(* CoDeSys 2.3.9.47 project: mqtt.pro *)
(* Libraries: C:\Program Files\WAGO Software\CoDeSys V2.3\Targets\WAGO\Libraries\32_Bit\oscat_basic_333.lib 9.2.16 17:15:54, SysLibSockets.lib 22.5.14 15:16:32, WagoLibEthernet_01.lib 11.2.16 17:05:44, Standard.lib 20.5.14 07:13:26, Iecsfc.lib 16.5.13 13:00:50, SYSLIBCALLBACK.LIB 16.5.13 13:00:50 *)

(* PLC configuration (modules and I/O channels)
K-Bus [K_Bus] node 0, in %IB0 out %QB0 {KbusBusMode = 1; KbusCycleTime = 10000; KbusThreadPriority = 0; KbusSetOutputsToZeroOnApplicationStop = 1}
Modbus variables [PFC200MODBUS] node 1, in %IB0 out %QB0 {PlcStopBehaviour = 1; FiledbusErrorBehaviour = 1; TcpOperation = 1; TcpPort = 502; TcpTimeout = 600; UdpOperation = 1; UdpPort = 502; RtuOperation = 0; NodeId = 1; ResponseTimeout = 5000; Interface = 0; Baud = 115200; StopBits = 1; Parity = 1; FlowCtrl = 0; PhysInterface = 0}
unused [PFC200CANOPEN_UNUSED] node 2, in %IB6000 out %QB6000
Modbus-Master [MB_MASTER] node 3, in %IB0 out %QB0
*)

(* Task configuration *)
TASK Schedule (PRIORITY := 31, INTERVAL := T#100ms);
	PLC_PRG();
END_TASK

(* Global variable list: Globale_Variablen *)
VAR_GLOBAL
	xxSubscribe: BOOL := TRUE;
	xxPublish : BOOL     := TRUE;
	SubPubState : INT;
END_VAR

(* Data type *)
TYPE Buffer :
STRUCT
	data : ARRAY [0..MAX_RECEIVE_TCP_CLIENT] OF BYTE;
	iPos : DWORD := 0;
END_STRUCT
END_TYPE

(* Data type *)
TYPE ConnectFlags :
STRUCT
	xUsername     : BOOL;
	xPassword     : BOOL;
	xWillRetain   : BOOL;
	xWillQoS1     : BOOL;
    xWillQoS2     : BOOL;
	xWillFlag     : BOOL;
	xCleanSession : BOOL;
END_STRUCT
END_TYPE

(* Data type *)
TYPE FixedHeader :
STRUCT
	bMessageType : BYTE := 16#00;
	xDUP_FLAG    : BOOL := FALSE;
	xQos         : BYTE := 16#00; (*0,1,2*)
	xRetain      : BOOL := FALSE;
END_STRUCT
END_TYPE

(* Data type *)
TYPE FixedHeaderSub :
STRUCT
	bMessageType : BYTE := 8;
	xReserved         : BYTE := 2;
END_STRUCT
END_TYPE

(* POU PLC_PRG, ST *)
PROGRAM PLC_PRG
VAR
	mqttClient: MQTT_Client;
	xPublish: BOOL;
	xSubscribe: BOOL;
END_VAR
mqttClient(
xPublish := xxPublish, (* I/O variable to publish to a TOPIC *)
xSubscribe := xxSubscribe,  (* NOT SUPPORTED, but must be here for I/O *)
sIP:='10.210.10.60', (* IP of the MQTT Broker *)
wPortNumber:=1883,  (* PORT of the MQTT Broker *)
(* AUTH: When no authentication is needed, leave the following fields Blank *)
sUsername:='',  (* Username to connect with the MQTT Broker *)
sPassword:='' (* password to connect with the MQTT Broker *)
);

mqttClient.sTopic := 'sub';
mqttClient.sQoS := 16#00;

mqttClient.pTopic := 'pub';
mqttClient.pQoS := 16#00;
mqttClient.pRetained := FALSE;
mqttClient.pPayload := 'wow';
END_PROGRAM

(* POU MQTT_Client, ST *)
FUNCTION_BLOCK MQTT_Client
VAR CONSTANT
	VERSION 	: BYTE := 16#03;
	Reserved   	: BYTE := 0;
	CONNECT     : BYTE := 1;
	CONNACK     : BYTE := 2;
	PUBLISH     : BYTE := 3;
	PUBACK      : BYTE := 4;
	PUBREC      : BYTE := 5;
	PUBREL      : BYTE := 6;
	PUBCOMP     : BYTE := 7;
	SUBSCRIBE   : BYTE := 8;
	SUBACK      : BYTE := 9;
	UNSUBSCRIBE : BYTE := 10;
	UNSUBACK    : BYTE := 11;
	PINGREQ     : BYTE := 12;
	PINGRESP    : BYTE := 13;
	DISCONNECT  : BYTE := 14;
	Reserved2   : BYTE := 15;

	CONNECTED   : INT := 30;
	NOT_CONNECTED: INT := 40;
	TIMEOUT : INT := 50;
	WAIT_RESPONSE : INT := 60;

	CONNECTION_TIMEOUT : TIME := t#10s;

	SUBSCRIBED : INT := 70;
	PUBLISHED : INT := 80;
	WAIT_RESPONSE_PUBLISH : INT := 90;
END_VAR

VAR
	fixedHeaderSub : BYTE;
	sendBuffer : Buffer;
	receiveBuffer : Buffer;
	fixedHeader: FixedHeader;
	variableHeader: Buffer;
	payLoad:  Buffer;
	connectFlags: ConnectFlags;
	tcpClient: TCP_Client;
	xTcpConnected: BOOL := FALSE;
	xStartSend: BOOL := FALSE;
	diReceiveCount: DINT;
	connectionTimer: TON;
	xTimeOut: BOOL;
	incomingMessageType: BYTE;
	eState: INT;
	xStartTimer: BOOL;

	a : Buffer;
	b : Buffer;
	i : DINT;
	publishDa : REAL;

	c : BOOL;
	(*xPublishTimeOut: BOOL;*)
END_VAR

VAR_INPUT
	sTopic: STRING;
	pTopic: STRING;
	pPayload: STRING;
	pRetained : BOOL;
	pQoS : BYTE;
	sQoS : BYTE;
	sIp : STRING;
	wPortNumber : WORD;
	sUsername : STRING;
	sPassword : STRING;
END_VAR

VAR_IN_OUT
	xPublish: BOOL;
	xSubscribe: BOOL;
END_VAR

VAR_OUTPUT
	xConnected : BOOL := FALSE;
	xBusy : BOOL := FALSE;
END_VAR
tcpClient.sIPaddress := sIp;
tcpClient.wPortNumber := wPortNumber;

tcpClient.ptSendData := ADR(sendBuffer.data);
tcpClient.diSendCount := sendBuffer.iPos;

tcpClient(xOpenConnection:=TRUE,
xStartSend:=xStartSend,
aReceiveBuffer := receiveBuffer.data,
diReceiveCount := diReceiveCount);

xTcpConnected := tcpClient.xConnected;
xBusy := xStartSend;

IF NOT xTcpConnected THEN
	eState := NOT_CONNECTED;
	xConnected := FALSE;
 	RETURN;
END_IF;

(* INIT *)
payLoad.iPos := 0;
variableHeader.iPos := 0;

connectionTimer(IN:=xStartTimer, PT:=CONNECTION_TIMEOUT-t#2s);
xTimeOut := connectionTimer.Q;

(*publishTimer(IN := xStartPublishTimer, PT := CONNECTION_TIMEOUT-t#5s);
xPublishTimeOut := publishTimer.Q;
(*Calculate redivelery*)
IF xPublishTimeOut THEN
END_IF*)


(* Calculate the current state *)
IF xTimeOut THEN
	eState := TIMEOUT;
ELSIF eState <> CONNECTED AND eState <> TIMEOUT AND eState <> WAIT_RESPONSE THEN
	eState := NOT_CONNECTED;
END_IF

(* Execute current state *)
CASE eState OF

CONNECTED:
	IF diReceiveCount <> 0 THEN
		incomingMessageType := receiveBuffer.data[0];
		IF incomingMessageType = SHL(PINGRESP, 4) THEN
			xStartTimer := TRUE;
		END_IF
		IF incomingMessageType = SHL(PUBLISH, 4)  THEN
			_ARRAY_INIT(ADR(a), SIZEOF(a), 0);
			FOR i:=0 TO diReceiveCount-1 BY 1 DO
				a.data[i] := receiveBuffer.data[i];
			END_FOR
		END_IF

		IF incomingMessageType = SHL(PUBACK, 4)  THEN
			_ARRAY_INIT(ADR(b), SIZEOF(b), 0);
			FOR i:=0 TO diReceiveCount-1 BY 1 DO
				b.data[i] := receiveBuffer.data[i];
			END_FOR
		END_IF

		diReceiveCount := 0;
	END_IF

	c := xxPublish AND xxSubscribe;
	IF   c   THEN
		SubPubState := SUBSCRIBED;
	ELSE
		SubPubState := PUBLISHED;
	END_IF;

	CASE SubPubState OF
			SUBSCRIBED:
				IF xxSubscribe THEN
					_BUFFER_CLEAR(ADR(sendBuffer), SIZEOF(sendBuffer));

					fixedHeaderSub :=  BYTE_OF_BIT(FALSE, TRUE, FALSE, FALSE, FALSE, FALSE, FALSE, TRUE); (*FIXED_HEADER*)
					(*fixedHeaderSub.bMessageType := SUBSCRIBE;*)

					_BUFFER_PUSH(ADR(variableHeader), 16#00);(* Message ID *)
					_BUFFER_PUSH(ADR(variableHeader), 16#00);

					_BUFFER_PUSH_STRING(ADR(payLoad), sTopic, TRUE);
					_BUFFER_PUSH(ADR(payLoad), sQoS); (*QoS 0 16#00*);

					sendBuffer.iPos := 0;
					CREATE_MESSAGE_SUB(ADR(sendBuffer), fixedHeaderSub, variableHeader, payLoad);

					xxSubscribe := FALSE;
					(**xxSubscribe := TRUE;**)
					xStartSend := TRUE;
					SubPubState := PUBLISHED;
				END_IF

			 PUBLISHED:
				IF xxPublish THEN
					fixedHeader.bMessageType := PUBLISH;
					fixedHeader.xDUP_FLAG := FALSE;
					(*fixedHeader.xQos := 16#00; (* only QoS 0 supported *)*)
					fixedHeader.xQoS := pQoS;
					fixedHeader.xRetain := pRetained;

					_BUFFER_PUSH_STRING(ADR(variableHeader), pTopic, TRUE); (* Topic *)
					IF fixedHeader.xQos > 16#00 THEN
						_BUFFER_PUSH(ADR(variableHeader), 16#00);(* Message ID *)
						_BUFFER_PUSH(ADR(variableHeader), 16#00);
					END_IF

					_BUFFER_PUSH_STRING(ADR(payLoad), pPayload, FALSE);

					sendBuffer.iPos := 0;
					CREATE_MESSAGE(ADR(sendBuffer), fixedHeader, variableHeader, payLoad);

					xxPublish := TRUE;
					xxSubscribe := TRUE;
					SubPubState := SUBSCRIBED;
					xStartSend := TRUE;
				END_IF
	END_CASE

NOT_CONNECTED:
	sendBuffer.iPos := 0;
	xStartTimer := FALSE;
	fixedHeader.bMessageType := CONNECT;

	_BUFFER_PUSH_STRING(ADR(variableHeader),'MQIsdp', TRUE); (* Protocol Name*)
	_BUFFER_PUSH(ADR(variableHeader), 3); (* Version Number*)

	connectFlags.xCleanSession := TRUE;
	connectFlags.xWillFlag     := FALSE;
	connectFlags.xWillQoS1     := FALSE;
	connectFlags.xWillQoS2     := FALSE;
	connectFlags.xWillRetain   := FALSE;
	IF LEN(sUsername) > 0 THEN
		connectFlags.xUsername := TRUE;
	ELSE
		connectFlags.xUsername := FALSE;
	END_IF
	IF LEN(sPassword) > 0 THEN
		connectFlags.xPassword := TRUE;
	ELSE
		connectFlags.xPassword := FALSE;
	END_IF

	_BUFFER_PUSH(ADR(variableHeader), BYTE_OF_BIT(FALSE,
															connectFlags.xCleanSession,
															connectFlags.xWillFlag,
															connectFlags.xWillQoS1,
															connectFlags.xWillQoS2,
															connectFlags.xWillRetain,
															connectFlags.xPassword,
															connectFlags.xUsername));

	_BUFFER_PUSH(ADR(variableHeader), 16#00);
	_BUFFER_PUSH(ADR(variableHeader), 16#0A); (* Keep Alive: 10s *)

	_BUFFER_PUSH_STRING(ADR(payload), 'PLC', TRUE); (* Client Identfier *)

	IF connectFlags.xUsername THEN
		_BUFFER_PUSH_STRING(ADR(payload), sUsername, TRUE); (* Username *)
	END_IF

	IF connectFlags.xPassword THEN
		_BUFFER_PUSH_STRING(ADR(payload), sPassword, TRUE); (* Password *)
	END_IF

	CREATE_MESSAGE(ADR(sendBuffer), fixedHeader, variableHeader, payLoad);

	eState := WAIT_RESPONSE;
	xStartSend := TRUE;

TIMEOUT:
	sendBuffer.iPos := 0;
	xStartTimer := FALSE;
	fixedHeader.bMessageType := PINGREQ;
	CREATE_MESSAGE(ADR(sendBuffer), fixedHeader, variableHeader, payLoad);

	eState := CONNECTED;
	xStartSend := TRUE;

WAIT_RESPONSE:
	incomingMessageType := receiveBuffer.data[0];
	IF incomingMessageType = SHL(CONNACK, 4) THEN
		(* TODO: Check return code *)
		xConnected := TRUE;
		xStartTimer := TRUE;
		eState := CONNECTED;
		diReceiveCount := 0;
	END_IF
END_CASE
END_FUNCTION_BLOCK

(* POU _BUFFER_PUSH, ST *)
FUNCTION _BUFFER_PUSH : BOOL
VAR_INPUT
	PT  : POINTER TO Buffer;
	IN  : BYTE;
END_VAR

VAR
END_VAR
(* pushed data to a buffer array *)
PT^.data[PT^.iPos] := IN;

PT^.iPos := PT^.iPos + 1;

_BUFFER_PUSH := TRUE;
END_FUNCTION

(* POU _BUFFER_PUSH_STRING, ST *)
FUNCTION _BUFFER_PUSH_STRING : BOOL
VAR_INPUT
	PT : POINTER TO Buffer;
	IN : STRING;
	INCLUDE_LENGTH : BOOL := FALSE;
END_VAR
VAR
	sPT : POINTER TO BYTE;
	iLen : DWORD;
	i : DWORD;
	nxtPtr: POINTER TO BYTE;
END_VAR
iLen := LEN(IN);
sPT := ADR(IN);

IF INCLUDE_LENGTH THEN
	_BUFFER_PUSH(PT, BYTE_OF_DWORD(iLen,1));
	_BUFFER_PUSH(PT, BYTE_OF_DWORD(iLen,0));
END_IF

FOR i:=0 TO iLen-1 BY 1 DO
	nxtPtr := sPT + i * SIZEOF(sPT^);
	_BUFFER_PUSH(PT, nxtPtr^);
END_FOR
END_FUNCTION

(* POU CREATE_MESSAGE_SUB, ST *)
FUNCTION CREATE_MESSAGE_SUB : BOOL
VAR_INPUT
	PT          			:POINTER TO Buffer;
	fixedHeader      	: BYTE;
	variableHeader  	:Buffer;
	payLoad         		:Buffer;
END_VAR
VAR
	bTemp  			:BYTE;
	remainingLength	:DWORD;
END_VAR
(* FIXED HEADER *)
(* BYTE 1 *)
(*bTemp := bTemp OR SHL(fixedHeader, 4);*)
(*bTemp := bTemp OR fixedHeader;*)
bTemp := fixedHeader;

_BUFFER_PUSH(PT, bTemp);

(* BYTE 2 *)
remainingLength := variableHeader.iPos + payLoad.iPos;

ENCODE_REMAINING_LENGTH(PT, remainingLength);
(*_BUFFER_PUSH(PT, remainingLength);*)

(* VARIABLE HEADER *)
_BUFFER_CONCAT(PT, ADR(variableHeader));

(* PAYLOAD *)
_BUFFER_CONCAT(PT, ADR(payLoad));
END_FUNCTION

(* POU ENCODE_REMAINING_LENGTH, ST *)
FUNCTION ENCODE_REMAINING_LENGTH : BOOL
VAR_INPUT
	PT : POINTER TO Buffer;
	LENGTH : DWORD;
END_VAR
VAR
	wPt : POINTER TO DWORD; (*4 bytes*)
	digit: DWORD;
	i: UINT;
END_VAR
wPt := ADR(LENGTH);

IF LENGTH = 0 THEN
	_BUFFER_PUSH(PT, 16#00);
	RETURN;
END_IF

WHILE LENGTH > 0 DO
	digit := LENGTH MOD 128;
	LENGTH := LENGTH / 128;
	
	IF LENGTH > 0 THEN
		digit := digit OR 16#80;
	END_IF
	_BUFFER_PUSH(PT, BYTE_OF_DWORD(digit,0));
END_WHILE
END_FUNCTION

(* POU _BUFFER_CONCAT, ST *)
FUNCTION _BUFFER_CONCAT : BOOL
VAR_INPUT
	PT  : POINTER TO Buffer;
	PTContact  : POINTER TO Buffer;
END_VAR
VAR
	i: INT;
END_VAR
FOR i:=0 TO DWORD_TO_INT(PTContact^.iPos) -1 BY 1 DO
	_BUFFER_PUSH(PT, PTContact^.data[i]);
END_FOR
END_FUNCTION

(* POU CREATE_MESSAGE, ST *)
FUNCTION CREATE_MESSAGE : BOOL
VAR_INPUT
	PT          : POINTER TO Buffer;
	fixedHeader     : FixedHeader;
	variableHeader  : Buffer;
	payLoad         : Buffer;
END_VAR
VAR
	bTemp  : BYTE;
	remainingLength: DWORD;
END_VAR
(* FIXED HEADER *)
(* BYTE 1 *)
bTemp := bTemp OR SHL(fixedHeader.bMessageType, 4) OR SHL(FixedHeader.xQos, 1);

BIT_LOAD_B(bTemp, FixedHeader.xDUP_FLAG, 3);
BIT_LOAD_B(bTemp, FixedHeader.xRetain, 0);

_BUFFER_PUSH(PT, bTemp);

(* BYTE 2 *)
remainingLength := variableHeader.iPos + payLoad.iPos;

ENCODE_REMAINING_LENGTH(PT, remainingLength);
(*_BUFFER_PUSH(PT, remainingLength);*)

(* VARIABLE HEADER *)
_BUFFER_CONCAT(PT, ADR(variableHeader));

(* PAYLOAD *)
_BUFFER_CONCAT(PT, ADR(payLoad));
END_FUNCTION

(* POU _BUFFER_SET, ST *)
FUNCTION _BUFFER_SET : BOOL
VAR_INPUT
	PT  : POINTER TO Buffer;
	IN  : BYTE;
	POS : UINT := 0;
END_VAR
VAR
END_VAR
PT^.data[POS] := IN;

IF PT^.iPos < POS THEN
	PT^.iPos := POS;
END_IF
END_FUNCTION
